PROGRAM MAIN
VAR
END_VAR

END_PROGRAM

(* stored: Version 1.1.0.1
   POU MAIN: Id {703308ff-0237-49b9-9852-9670b2ad865e} *)
